TYPE ST_ReadConvDb :
STRUCT
	nId			: DINT;
	sMachine	: STRING(20);
	sWorkpiece	: STRING(20);
	dtTimestart	: DT;
	dtTimestop	: DT;
	sDuration	: STRING(255); // interval data type not supported
END_STRUCT
END_TYPE

(* stored: Version 1.1.0.1
   DUT ST_ReadConvDb: Id {3aeea6be-4d0a-49e3-b992-ca8ddb54615f} *)
